DATA_BLOCK "DB_G16StatusModel"
{ S7_Optimized_Access := 'TRUE' }
VERSION : 0.1
NON_RETAIN
   VAR
      Data : "UDT_G16StatusModel";
   END_VAR

BEGIN
END_DATA_BLOCK
